Yaskawa INFORM job: ROVI_RESET.JBI

/JOB
//NAME ROVI_RESET
///FOLDERNAME ROVI
//POS
///NPOS 0,0,0,0,0,0
//INST
///DATE 2019/12/05 14:48
///ATTR SC,RW
///GROUP1 RB1
NOP
SET B080 0
WAIT B080=255
RET I080
END
